FUNCTION_BLOCK FB_Mover IMPLEMENTS IObject
VAR_INPUT
END_VAR
VAR_OUTPUT
END_VAR
VAR
    _ID           : INT;                           // hard id number of the mover
    _MoverAxis    : REFERENCE TO FB_SimuMoverAxis; // reference to an FB_SimuMoverAxis
    _AttachedTool : REFERENCE TO FB_PieceHolder;   // attached toolhead
    _Station      : REFERENCE TO FB_Station;       // current station

    _State : MoverState_e := MoverState_e.WaitOnNextStation; // current mover state
	
	_iID : INT := 0; // instance ID, is set during FB_Init using the value of _iInstanceCounter 
END_VAR
VAR CONSTANT
END_VAR
VAR_STAT
	_iInstanceCounter : INT := 1; // instance counter
END_VAR

PROPERTY AttachedPieceHolder : REFERENCE TO FB_PieceHolder
GET
AttachedPieceHolder REF=_AttachedTool;
END_GET
SET
_AttachedTool REF= AttachedPieceHolder;
END_SET
END_PROPERTY

METHOD Equals : BOOL
VAR_INPUT
    object : ANY;
END_VAR
Equals := THIS = object.pValue;
END_METHOD

METHOD FB_init : BOOL
VAR_INPUT
    bInitRetains : BOOL; // if TRUE, the retain variables are initialized (warm start / cold start)
    bInCopyCode  : BOOL; // if TRUE, the instance afterwards gets moved into the copy code (online change)
    ID           : INT;  // hard id number of the mover

    MoverAxis : REFERENCE TO FB_SimuMoverAxis; // reference to an FB_SimuMoverAxis
END_VAR
THIS^._iID := THIS^._iInstanceCounter;
THIS^._iInstanceCounter := THIS^._iInstanceCounter +1;
THIS^._ID := ID;
THIS^._MoverAxis REF= MoverAxis;
THIS^._AttachedTool REF=0;
THIS^._Station REF=0;
END_METHOD

// Is this mover behind a given position?
// this method do the opposit as IsInFront
METHOD IsBehind : BOOL
VAR_INPUT
    lrPosition : LREAL; // position to test
END_VAR
IsBehind := lrPosition > THIS^._MoverAxis.CurrentPos;
END_METHOD

// Is this mover is in front of a given position?
// Use this function also to check if the next station is behind the mover or not.
// In this case, the mover needs to complet its turn for accessing the given station
METHOD IsInFront : BOOL
VAR_INPUT
    lrPosition : LREAL; // position to test
END_VAR
IsInFront := lrPosition < THIS^._MoverAxis.CurrentPos;
END_METHOD

METHOD IsInStationPos : BOOL
VAR_INPUT
END_VAR
// we have to substract the piecholder offset to find the station position again
IF CONST.BIND_WITH_TRACK THEN
    IsInStationPos :=
        THIS^.Station.Position.isInPos(gMoverAxis.I_CT_Shuttle_from_BR.asStruct[THIS^._ID].diCurrentPos_um / 1000 -
                                       THIS^._AttachedTool.PosOffset -
                                       THIS^.Station.Offset);
ELSE
    IsInStationPos := THIS^.Station.Position
        .isInPos(THIS^.MoverAxis.CurrentPos - THIS^._AttachedTool.PosOffset - THIS^.Station.Offset);
END_IF
END_METHOD

PROPERTY MoverAxis : REFERENCE TO FB_SimuMoverAxis
GET
MoverAxis REF= _MoverAxis;
END_GET
SET
_MoverAxis REF= MoverAxis;
END_SET
END_PROPERTY

// Move to the current set station. Can only move if the current process are running
METHOD MoveToStation : REFERENCE TO FB_Mover
VAR_INPUT
END_VAR
IF THIS^._State <> MoverState_e.InOperation THEN
    THIS^.MoverAxis.MoveTo(TO_POS(THIS^.Station.Position.lrWorkPosition + THIS^._AttachedTool.PosOffset + THIS^.Station.Offset));
    THIS^._State := MoverState_e.MovingToStation;
END_IF

MoveToStation REF= THIS^;
END_METHOD

// Move to waiting spot
// The mover will not move if the waiting spot can not store
// a full mover
METHOD MoveToWaitSpot : REFERENCE TO FB_Mover
VAR_INPUT
END_VAR
IF THIS^._State <> MoverState_e.InOperation THEN
    IF THIS^.Station.WaitPos <= (THIS^.Station.Position.lrWorkPosition - CONST.MAX_MOVER_SIZE) THEN
        THIS^.MoverAxis.MoveTo(TO_POS(THIS^.Station.WaitPos + THIS^._AttachedTool.PosOffset + THIS^.Station.Offset));
    END_IF
END_IF

THIS^._State := MoverState_e.MovingToStation;

MoveToWaitSpot REF= THIS^;
END_METHOD

// Set a specic piece holder. This will affect the station position offset
METHOD SetPieceHolder : REFERENCE TO FB_Mover
VAR_INPUT
	pieceHolder : REFERENCE TO FB_PieceHolder;
END_VAR
IF __ISVALIDREF(pieceHolder) THEN
	THIS^._AttachedTool REF=pieceHolder;
END_IF
SetPieceHolder REF= THIS^;
END_METHOD

// Set the next station of the mover. This action does not make the mover moves. 
// First you need to set the station. Then, depending on the station scenario,
// you will run to it when its current process is finished or move to it
// as quick as possible
METHOD SetStation : REFERENCE TO FB_Mover
VAR_INPUT
	Station : REFERENCE TO FB_Station;
END_VAR
IF __ISVALIDREF(Station) AND_THEN (THIS^._State <> MoverState_e.InOperation) THEN
    THIS^._Station REF= Station;
    THIS^._State   := MoverState_e.WaitOnNextStation;
ELSE
    ASSERT(0);
END_IF

SetStation REF= THIS^;
END_METHOD

PROPERTY State : MoverState_e
GET
State := _State;
END_GET
SET
_State := State;
END_SET
END_PROPERTY

PROPERTY Station : REFERENCE TO FB_Station
GET
Station REF=_Station;
END_GET
SET
_Station REF=Station;
END_SET
END_PROPERTY

// take a position and return always a positive integer between 0 and MAX_TRACK_LENGTH
METHOD PRIVATE TO_POS : DINT
VAR_INPUT
	pos : LREAL;
END_VAR
IF pos < 0 THEN
    TO_POS := LREAL_TO_DINT(pos + CONST.MAX_TRACK_LENGTH);

ELSIF pos >= CONST.MAX_TRACK_LENGTH THEN
    TO_POS := LREAL_TO_DINT(pos) MOD LREAL_TO_DINT(CONST.MAX_TRACK_LENGTH);

ELSE
    TO_POS := LREAL_TO_DINT(pos);

END_IF
END_METHOD

METHOD ToString : STRING
VAR_INPUT
END_VAR
ToString := CONCAT('FB_Mover_', TO_STRING(THIS^._iID));
END_METHOD

END_FUNCTION_BLOCK

(* stored: Version 1.1.0.1, ProductVersion 3.1.4024.6
   POU FB_Mover: Id {147d877f-8a39-46b8-8ff1-e23190be69f7}, SpecialFunc None
   Property AttachedPieceHolder: Id {1f1520b6-17b9-443d-9101-58c2158353cb}
   Get Get: Id {7bc424cc-e238-4415-b174-26b9a1b9bd88}
   Set Set: Id {b3043ba1-5edb-429d-81cb-c6094b6860ba}
   Method Equals: Id {f14740f4-58b8-4c64-8940-c4b242e3aa11}
   Method FB_init: Id {f1ad25b4-41be-48ac-a3cf-a51a38b48b2b}
   Method IsBehind: Id {1364b0b6-81a4-4545-a8c6-935b8f76ea04}
   Method IsInFront: Id {42e385d9-249e-426b-a8a4-bd8bc25cd49a}
   Method IsInStationPos: Id {8f1d1c8f-d3a0-4e9f-9fe0-8845545f2ce3}
   Property MoverAxis: Id {667c64f3-25b7-4e93-87f1-34db05ea3af9}
   Get Get: Id {c2459c87-114e-4ec7-b3db-caf985555ebd}
   Set Set: Id {05348f58-2bb4-4f7f-8f83-3865d24f3ec6}
   Method MoveToStation: Id {eca588ef-140f-424d-b8d0-9320c30f98a1}
   Method MoveToWaitSpot: Id {e6a96abf-85ca-4700-ac8c-39eb7eb170c8}
   Method SetPieceHolder: Id {3656c226-034e-4545-af0f-2c2902573b50}
   Method SetStation: Id {99a6cded-9b90-4798-b54e-b9966cee1bc2}
   Property State: Id {450dea2c-6489-4063-a805-699ccf8a7f48}
   Get Get: Id {a0133e0b-8f6e-4d2b-81b4-55f4faaae79f}
   Set Set: Id {b22fe45a-1d49-466d-bfcd-05811e0eef14}
   Property Station: Id {7bbd8745-ad21-4808-9c00-2034901cee36}
   Get Get: Id {c1123c17-aefe-44e5-a428-dc0f7f2b27ab}
   Set Set: Id {2c75b98f-8c6d-40fc-a63d-e74234713015}
   Method TO_POS: Id {0a18dcda-f783-4400-9438-3adfacc7213c}
   Method ToString: Id {54c07018-71f2-4cf5-9d31-ef8ca5167ad0} *)
